{attribute 'hide'}
PROGRAM General_TestSuite
VAR
	anyToStringTest : AnyToString_Test;
	isValueEvenTest : IsValueEven_Test;
	longStringLenTest : LongStringLen_Test;
END_VAR

END_PROGRAM

(* stored: Version 1.1.0.1, ProductVersion 3.1.4024.9
   POU General_TestSuite: Id {3f2929a5-2d3e-46f3-a12c-f11259cd13c1}, SpecialFunc None *)
